Fanuc KAREL source: kb00097.KL

-- PROVISIONAL review KL for V940-1; original PC SHA256 e63435e548b3c550a4f264d6ee933e708fd51e2e8cf0cd6a2ac053e41d15c0db
-- Incomplete behavior may be omitted. Consult companion uncertainty JSON. Do not deploy.
PROGRAM KB00097
%NOLOCKGROUP
BEGIN
  -- V9_ZERO_TABLE_METADATA_HINT layout=0002_ascii; no indexed target words; source/name/runtime held
  -- UNRESOLVED_PC offsets 5-14; opcodes 3F,75
  -- UNRESOLVED_PC offsets 19-26; opcodes 9D,23
  -- UNRESOLVED_PC offsets 31-38; opcodes 9D,23
  -- UNRESOLVED_PC offsets 43-50; opcodes 9D,23
  -- UNRESOLVED_PC offsets 55-64; opcodes 3F,75
  -- UNRESOLVED_PC offsets 69-76; opcodes 9D,23
  -- UNRESOLVED_PC offsets 81-125; opcodes 27,22,2A,22,22,22,22,2A,22,31
  -- UNRESOLVED_PC offsets 130-134; opcodes 7F
END KB00097
